FUNCTION_BLOCK FB_FakeBaseUnit IMPLEMENTS I_BaseUnit

END_FUNCTION_BLOCK

(* stored: Version 1.1.0.1, ProductVersion 3.1.4026.18
   POU FB_FakeBaseUnit: Id {2b467136-4428-4bb8-8923-6813cdc7ce02}, SpecialFunc None *)
